FUNCTION_BLOCK FB_ReadInput
VAR_INPUT
	rawInput	:	stRawInput;
END_VAR
VAR_IN_OUT
	input	:	stInput;
END_VAR
VAR
	tpStart	:	TP();
	tpAck	:	TP();
END_VAR

// temporizzatori a impulso per start e ack
	tpStart(IN := rawInput.Start, PT := T#200MS);
	tpAck(IN := rawInput.Ack, PT := T#200MS);

// aggiornamento ingressi virtuali
	input.start := tpStart.Q;
	input.stop := rawInput.Stop;
	input.ack := tpAck.Q;
	input.emg := rawInput.Emg;
	input.FC1 := rawInput.FC1;
	input.FC2 := rawInput.FC2;

END_FUNCTION_BLOCK

(* stored: Version 1.1.0.1
   POU FB_ReadInput: Id {78c7b48a-8a10-0503-2425-624957aba7fa}, SpecialFunc None *)
